FUNCTION_BLOCK FB_ADS_Read
VAR
	intState: INT;
	fbADSRDWRT: ADSRDWRT;
	Timer1: TON;
END_VAR
VAR_INPUT
	udintWriteLength:UDINT;
	udintReadLength:UDINT;
	dwSourceAddr:pvoid;
	dwDestAddr:PVOID;
	strNetID: STRING;
	timeReadDelay:TIME;
END_VAR
VAR_OUTPUT
	mADSError: BOOL;
	strADSErrorText: STRING;
END_VAR

timeReadDelay := LIMIT(T#100MS,timeReadDelay,T#24H);

CASE intState OF
	0:	(* start reading *)
		fbADSRDWRT.WRITELEN:=udintWriteLength;
		fbADSRDWRT.READLEN:=udintReadLength;
		fbADSRDWRT.SRCADDR:=dwSourceAddr;
		fbADSRDWRT.DESTADDR:=dwDestAddr;
		fbADSRDWRT.WRTRD:=TRUE;
		intState:=1000;
	1000: (* wait for reply *)
		IF NOT fbADSRDWRT.BUSY THEN
			fbADSRDWRT.WRTRD:=FALSE;
			IF NOT fbADSRDWRT.ERR THEN
				strADSErrorText:='no error';
				mADSError:=FALSE;
				Timer1.IN:=TRUE;
				intState:=1100;
			ELSE
				strADSErrorText:=F_AdsErrorText(fbADSRDWRT.ERRID);
				mADSError:=TRUE;
				Timer1.IN:=TRUE;
				intState:=1100;
			END_IF
		END_IF
	1100: (* wait to hold state *)
		fbADSRDWRT.WRTRD:=FALSE;
		IF Timer1.Q THEN
			Timer1.IN:=FALSE;
			intState:=0;
		END_IF
		
END_CASE

Timer1(PT:=timeReadDelay);


fbADSRDWRT(
	NETID:=strNetID,
	PORT:=851,
	IDXGRP:=16#F004,
	IDXOFFS:=0,
	TMOUT:=t#10s);


(*
VAR_INPUT
        NETID           : T_AmsNetId;
        PORT            : T_AmsPort;
        IDXGRP          : UDINT;
        IDXOFFS         : UDINT;
        WRITELEN                : UDINT;
        READLEN         : UDINT;
        SRCADDR                 : DWORD;
        DESTADDR                : DWORD;
        WRTRD           : BOOL;
        TMOUT           : TIME;
END_VAR
VAR_OUTPUT
        BUSY            : BOOL;
        ERR             : BOOL;
        ERRID           : UDINT;
END_VAR

*)

END_FUNCTION_BLOCK

(* stored: Version 1.1.0.1, ProductVersion 3.1.4024.12
   POU FB_ADS_Read: Id {53744c82-4d9c-4c0d-b285-44bc7613e791}, SpecialFunc None *)
